FUNCTION_BLOCK FB_ControlerDeviation
VAR_INPUT
	rCV : REAL;
	rPV : REAL;
	rMax : REAL;
	rTh : REAL;
END_VAR
VAR_OUTPUT
	bResult : real;
END_VAR
VAR
END_VAR

bResult := 0;
IF rMax <> 0 THEN
	bResult := ABS(rPV - rCV)/rMax;
END_IF

END_FUNCTION_BLOCK

(* stored: Version 1.1.0.1, ProductVersion 3.1.4026.12
   POU FB_ControlerDeviation: Id {ade406ed-6bac-45e6-9b2e-b0a1013e2d37}, SpecialFunc None *)
